TYPE "PLCtoMES_Common_ext"
VERSION : 0.1
   STRUCT
      "P-HeartBeat" : Bool;
   END_STRUCT;

END_TYPE

